Fanuc KAREL source: IO0069.KL

-- PROVISIONAL review KL for V940-1; original PC SHA256 d8689b940f867f41513b0c79bc9bb613b06b42f186ac068f703af3443cebb81f
-- Incomplete behavior may be omitted. Consult companion uncertainty JSON. Do not deploy.
PROGRAM IO0069
%NOLOCKGROUP
-- UNRESOLVED_LOCAL_POOL 5 cells at code offset 13; source declarations unknown
-- DIRECT_LOCAL_WORD_ACCESS alone does not prove INTEGER, REAL, or BOOLEAN
BEGIN
  -- V9_EXPOSED_INDEXED_TABLE_HINT layout=0001; 1 counted words exposed once; source arms/runtime held
  -- V9_ZERO_GLOBAL_LAYOUT_HINT count-one $GROUP table, zero relocation slots, two routine descriptors; executable preamble and source held
  -- V9_ANALOG_RDI_SIGNAL_HINT AIN condition constant_17
  -- UNRESOLVED_PC offsets 0-18; opcodes 2B,2C,7B
  -- UNRESOLVED_PC offsets 23-30; opcodes 9D,23
  -- UNRESOLVED_PC offsets 35-49; opcodes 2E,22,9D,33,35
  -- UNRESOLVED_PC offsets 54-61; opcodes 9D,23
  -- UNRESOLVED_PC offsets 66-77; opcodes 2E,23
  -- UNRESOLVED_PC offsets 82-96; opcodes 2E,19,9C,5B,79
  -- UNRESOLVED_PC offsets 101-115; opcodes 21,9D,52,23
  -- UNRESOLVED_PC offsets 125-129; opcodes 7F
  -- UNRESOLVED_PC offsets 134-138; opcodes 27,AA
  -- UNRESOLVED_PC offsets 143-147; opcodes 7F
END IO0069
